// Mitsubishi GX Works2 project: LABB1.2   PLC: FX3U/FX3UC

// global labels: Global1
VAR_GLOBAL
  VK_VAN1 AT X000 : BOOL;  (* VÅNINGSKNAPP *)
  VK_VAN2 AT X001 : BOOL;
  VK_VAN3 AT X002 : BOOL;
  VK_VAN4 AT X003 : BOOL;
  GL_VAN1 AT X004 : BOOL;  (* POSITIONSREGISTER *)
  GL_VAN2 AT X005 : BOOL;
  GL_VAN3 AT X006 : BOOL;
  GL_VAN4 AT X007 : BOOL;
  HK_VAN1 AT X010 : BOOL;
  HK_VAN2 AT X011 : BOOL;  (* HISSKNAPP *)
  HK_VAN3 AT X012 : BOOL;
  HK_VAN4 AT X013 : BOOL;
  HL_VAN1 AT Y000 : BOOL;  (* HISSLAMPA *)
  HL_VAN2 AT Y001 : BOOL;
  HL_VAN3 AT Y002 : BOOL;
  HL_VAN4 AT Y003 : BOOL;
  VL_VAN1 AT Y004 : BOOL;  (* VÅNINGSLAMPA *)
  VL_VAN2 AT Y005 : BOOL;
  VL_VAN3 AT Y006 : BOOL;
  VL_VAN4 AT Y007 : BOOL;
  Motor_upp AT Y010 : BOOL;  (* HISS UPP *)
  Motor_ner AT Y011 : BOOL;  (* HISS NER *)
  PULS_1Hz AT M8013 : BOOL;  (* KLOCKFREKVENS FÖR VL *)
  ALARM_10Hz AT M8012 : BOOL;  (* ALARMFREKVENS *)
  TEMP AT Y012 : BOOL;  (* TEMP *)
  SWITCH AT Y013 : BOOL;  (* SWITCH *)
  SEC AT D100 : INT;
  MINUTE AT D101 : INT;
  TIMMAR AT D102 : INT;
  DAG AT D103 : INT;
  MANAD AT D104 : INT;
  AR AT D105 : INT;
  SEC2 AT D110 : INT;
  MINUTE2 AT D111 : INT;
  TIMMAR2 AT D112 : INT;
  DAG2 AT D113 : INT;
  MANAD2 AT D114 : INT;
  AR2 AT D115 : INT;
END_VAR

PROGRAM MAIN
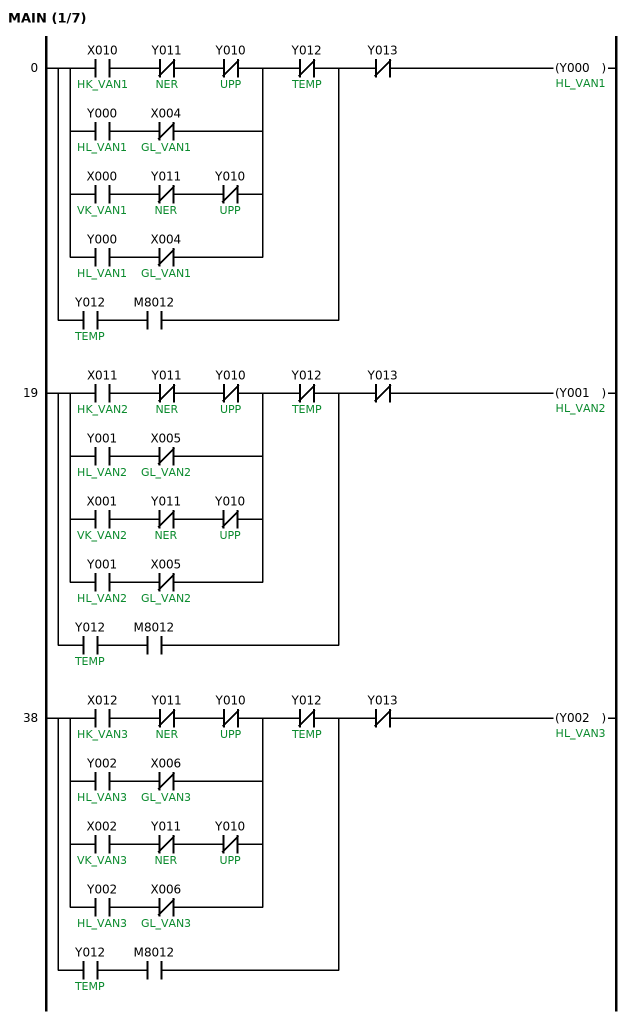
0     LD      X010  ; HK_VAN1
      ANI     Y011  ; NER
      ANI     Y010  ; UPP
      LD      Y000  ; HL_VAN1
      ANI     X004  ; GL_VAN1
      ORB
      LD      X000  ; VK_VAN1
      ANI     Y011  ; NER
      ANI     Y010  ; UPP
      ORB
      LD      Y000  ; HL_VAN1
      ANI     X004  ; GL_VAN1
      ORB
      ANI     Y012  ; TEMP
      LD      Y012  ; TEMP
      AND     M8012
      ORB
      ANI     Y013
      OUT     Y000  ; HL_VAN1
19    LD      X011  ; HK_VAN2
      ANI     Y011  ; NER
      ANI     Y010  ; UPP
      LD      Y001  ; HL_VAN2
      ANI     X005  ; GL_VAN2
      ORB
      LD      X001  ; VK_VAN2
      ANI     Y011  ; NER
      ANI     Y010  ; UPP
      ORB
      LD      Y001  ; HL_VAN2
      ANI     X005  ; GL_VAN2
      ORB
      ANI     Y012  ; TEMP
      LD      Y012  ; TEMP
      AND     M8012
      ORB
      ANI     Y013
      OUT     Y001  ; HL_VAN2
38    LD      X012  ; HK_VAN3
      ANI     Y011  ; NER
      ANI     Y010  ; UPP
      LD      Y002  ; HL_VAN3
      ANI     X006  ; GL_VAN3
      ORB
      LD      X002  ; VK_VAN3
      ANI     Y011  ; NER
      ANI     Y010  ; UPP
      ORB
      LD      Y002  ; HL_VAN3
      ANI     X006  ; GL_VAN3
      ORB
      ANI     Y012  ; TEMP
      LD      Y012  ; TEMP
      AND     M8012
      ORB
      ANI     Y013
      OUT     Y002  ; HL_VAN3
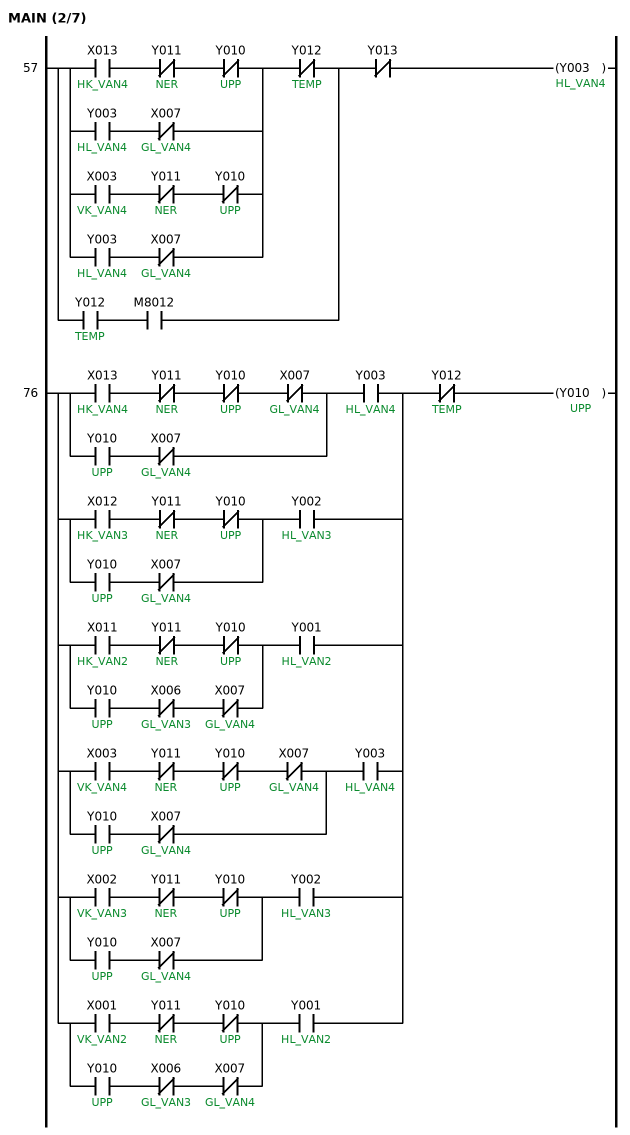
57    LD      X013  ; HK_VAN4
      ANI     Y011  ; NER
      ANI     Y010  ; UPP
      LD      Y003  ; HL_VAN4
      ANI     X007  ; GL_VAN4
      ORB
      LD      X003  ; VK_VAN4
      ANI     Y011  ; NER
      ANI     Y010  ; UPP
      ORB
      LD      Y003  ; HL_VAN4
      ANI     X007  ; GL_VAN4
      ORB
      ANI     Y012  ; TEMP
      LD      Y012  ; TEMP
      AND     M8012
      ORB
      ANI     Y013
      OUT     Y003  ; HL_VAN4
76    LD      X013  ; HK_VAN4
      ANI     Y011  ; NER
      ANI     Y010  ; UPP
      ANI     X007  ; GL_VAN4
      LD      Y010  ; UPP
      ANI     X007  ; GL_VAN4
      ORB
      AND     Y003  ; HL_VAN4
      LD      X012  ; HK_VAN3
      ANI     Y011  ; NER
      ANI     Y010  ; UPP
      LD      Y010  ; UPP
      ANI     X007  ; GL_VAN4
      ORB
      AND     Y002  ; HL_VAN3
      ORB
      LD      X011  ; HK_VAN2
      ANI     Y011  ; NER
      ANI     Y010  ; UPP
      LD      Y010  ; UPP
      ANI     X006  ; GL_VAN3
      ANI     X007  ; GL_VAN4
      ORB
      AND     Y001  ; HL_VAN2
      ORB
      LD      X003  ; VK_VAN4
      ANI     Y011  ; NER
      ANI     Y010  ; UPP
      ANI     X007  ; GL_VAN4
      LD      Y010  ; UPP
      ANI     X007  ; GL_VAN4
      ORB
      AND     Y003  ; HL_VAN4
      ORB
      LD      X002  ; VK_VAN3
      ANI     Y011  ; NER
      ANI     Y010  ; UPP
      LD      Y010  ; UPP
      ANI     X007  ; GL_VAN4
      ORB
      AND     Y002  ; HL_VAN3
      ORB
      LD      X001  ; VK_VAN2
      ANI     Y011  ; NER
      ANI     Y010  ; UPP
      LD      Y010  ; UPP
      ANI     X006  ; GL_VAN3
      ANI     X007  ; GL_VAN4
      ORB
      AND     Y001  ; HL_VAN2
      ORB
      ANI     Y012  ; TEMP
      OUT     Y010  ; UPP
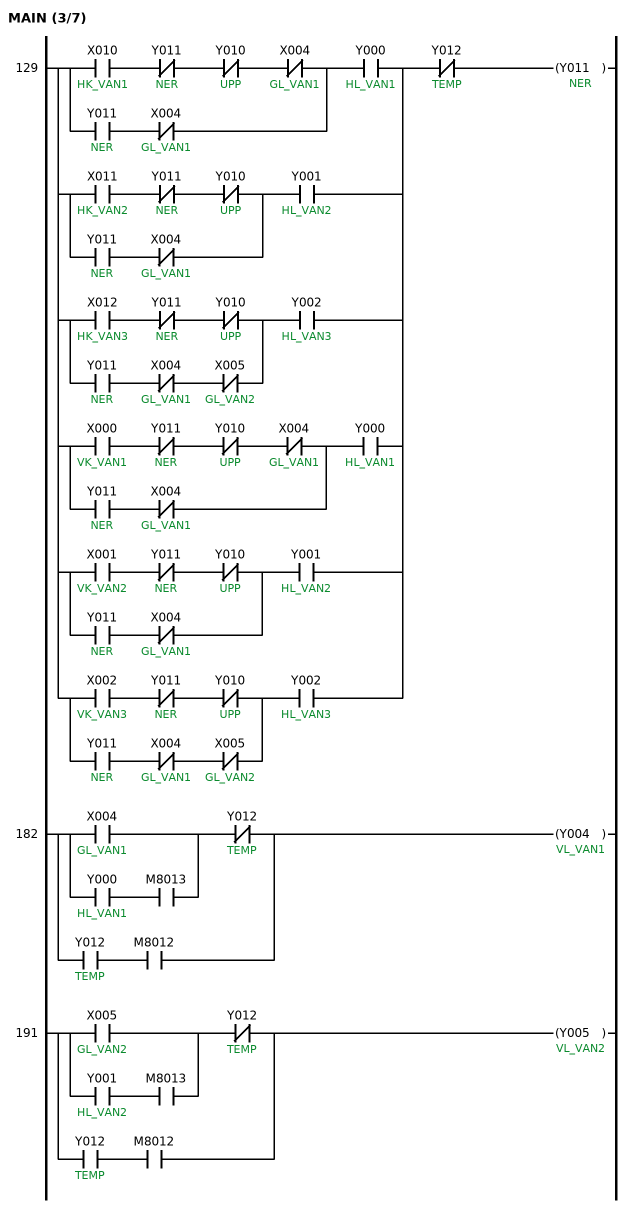
129   LD      X010  ; HK_VAN1
      ANI     Y011  ; NER
      ANI     Y010  ; UPP
      ANI     X004  ; GL_VAN1
      LD      Y011  ; NER
      ANI     X004  ; GL_VAN1
      ORB
      AND     Y000  ; HL_VAN1
      LD      X011  ; HK_VAN2
      ANI     Y011  ; NER
      ANI     Y010  ; UPP
      LD      Y011  ; NER
      ANI     X004  ; GL_VAN1
      ORB
      AND     Y001  ; HL_VAN2
      ORB
      LD      X012  ; HK_VAN3
      ANI     Y011  ; NER
      ANI     Y010  ; UPP
      LD      Y011  ; NER
      ANI     X004  ; GL_VAN1
      ANI     X005  ; GL_VAN2
      ORB
      AND     Y002  ; HL_VAN3
      ORB
      LD      X000  ; VK_VAN1
      ANI     Y011  ; NER
      ANI     Y010  ; UPP
      ANI     X004  ; GL_VAN1
      LD      Y011  ; NER
      ANI     X004  ; GL_VAN1
      ORB
      AND     Y000  ; HL_VAN1
      ORB
      LD      X001  ; VK_VAN2
      ANI     Y011  ; NER
      ANI     Y010  ; UPP
      LD      Y011  ; NER
      ANI     X004  ; GL_VAN1
      ORB
      AND     Y001  ; HL_VAN2
      ORB
      LD      X002  ; VK_VAN3
      ANI     Y011  ; NER
      ANI     Y010  ; UPP
      LD      Y011  ; NER
      ANI     X004  ; GL_VAN1
      ANI     X005  ; GL_VAN2
      ORB
      AND     Y002  ; HL_VAN3
      ORB
      ANI     Y012  ; TEMP
      OUT     Y011  ; NER
182   LD      X004  ; GL_VAN1
      LD      Y000  ; HL_VAN1
      AND     M8013
      ORB
      ANI     Y012  ; TEMP
      LD      Y012  ; TEMP
      AND     M8012
      ORB
      OUT     Y004  ; VL_VAN1
191   LD      X005  ; GL_VAN2
      LD      Y001  ; HL_VAN2
      AND     M8013
      ORB
      ANI     Y012  ; TEMP
      LD      Y012  ; TEMP
      AND     M8012
      ORB
      OUT     Y005  ; VL_VAN2
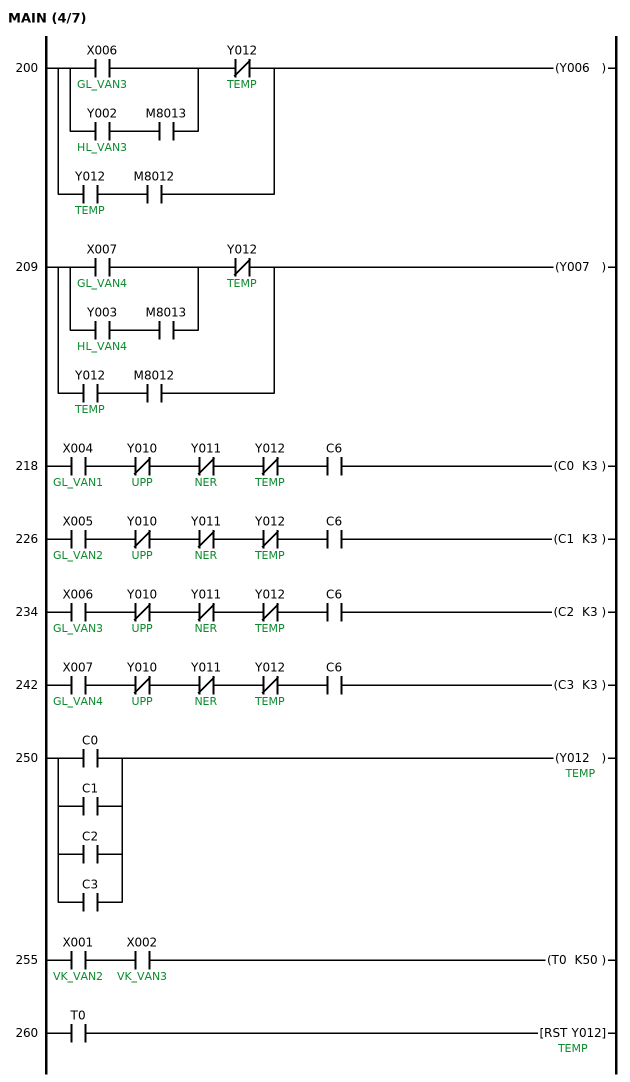
200   LD      X006  ; GL_VAN3
      LD      Y002  ; HL_VAN3
      AND     M8013
      ORB
      ANI     Y012  ; TEMP
      LD      Y012  ; TEMP
      AND     M8012
      ORB
      OUT     Y006
209   LD      X007  ; GL_VAN4
      LD      Y003  ; HL_VAN4
      AND     M8013
      ORB
      ANI     Y012  ; TEMP
      LD      Y012  ; TEMP
      AND     M8012
      ORB
      OUT     Y007
218   LD      X004  ; GL_VAN1
      ANI     Y010  ; UPP
      ANI     Y011  ; NER
      ANI     Y012  ; TEMP
      AND     C6
      OUT     C0 K3
226   LD      X005  ; GL_VAN2
      ANI     Y010  ; UPP
      ANI     Y011  ; NER
      ANI     Y012  ; TEMP
      AND     C6
      OUT     C1 K3
234   LD      X006  ; GL_VAN3
      ANI     Y010  ; UPP
      ANI     Y011  ; NER
      ANI     Y012  ; TEMP
      AND     C6
      OUT     C2 K3
242   LD      X007  ; GL_VAN4
      ANI     Y010  ; UPP
      ANI     Y011  ; NER
      ANI     Y012  ; TEMP
      AND     C6
      OUT     C3 K3
250   LD      C0
      OR      C1
      OR      C2
      OR      C3
      OUT     Y012  ; TEMP
255   LD      X001  ; VK_VAN2
      AND     X002  ; VK_VAN3
      OUT     T0 K50
260   LD      T0
      RST     Y012  ; TEMP
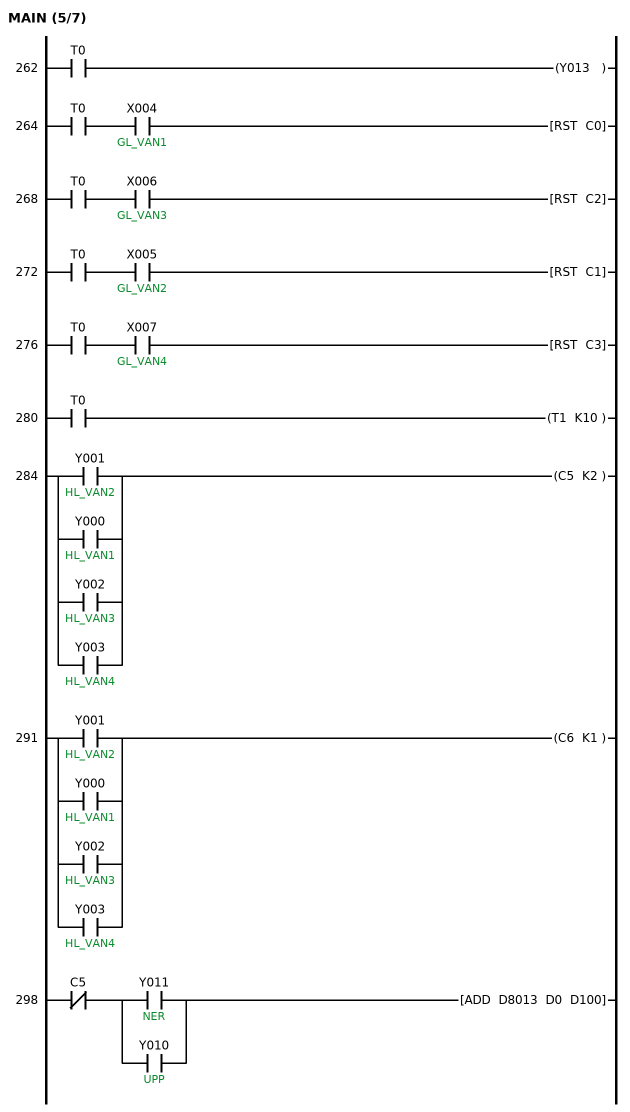
262   LD      T0
      OUT     Y013
264   LD      T0
      AND     X004  ; GL_VAN1
      RST     C0
268   LD      T0
      AND     X006  ; GL_VAN3
      RST     C2
272   LD      T0
      AND     X005  ; GL_VAN2
      RST     C1
276   LD      T0
      AND     X007  ; GL_VAN4
      RST     C3
280   LD      T0
      OUT     T1 K10
284   LD      Y001  ; HL_VAN2
      OR      Y000  ; HL_VAN1
      OR      Y002  ; HL_VAN3
      OR      Y003  ; HL_VAN4
      OUT     C5 K2
291   LD      Y001  ; HL_VAN2
      OR      Y000  ; HL_VAN1
      OR      Y002  ; HL_VAN3
      OR      Y003  ; HL_VAN4
      OUT     C6 K1
298   LDI     C5
      LD      Y011  ; NER
      OR      Y010  ; UPP
      ANB
      ADD     D8013 D0 D100
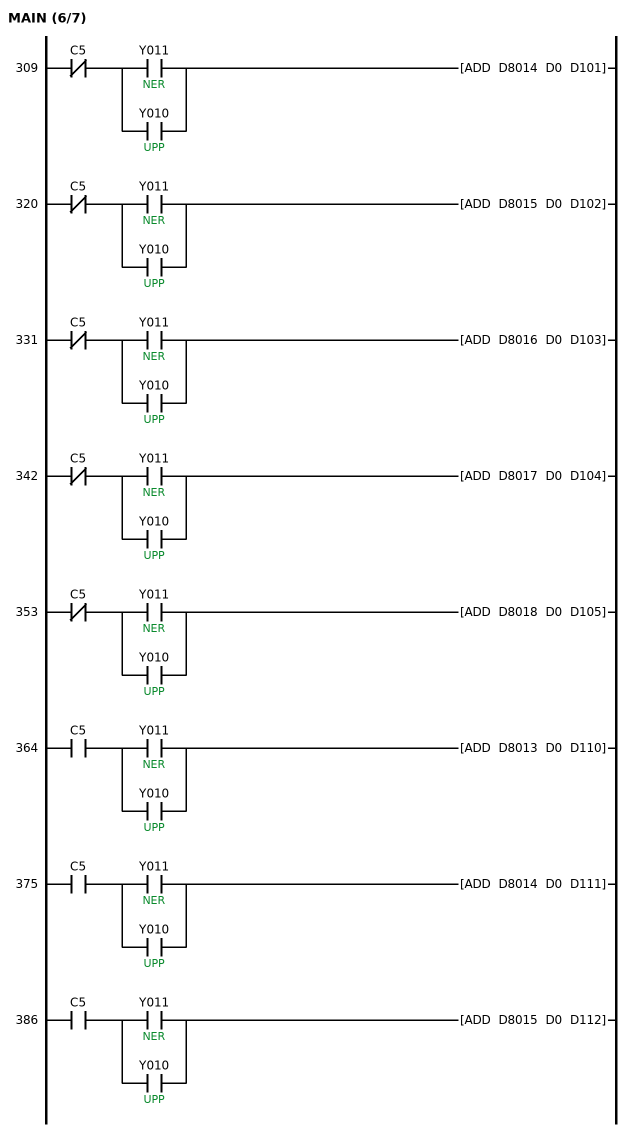
309   LDI     C5
      LD      Y011  ; NER
      OR      Y010  ; UPP
      ANB
      ADD     D8014 D0 D101
320   LDI     C5
      LD      Y011  ; NER
      OR      Y010  ; UPP
      ANB
      ADD     D8015 D0 D102
331   LDI     C5
      LD      Y011  ; NER
      OR      Y010  ; UPP
      ANB
      ADD     D8016 D0 D103
342   LDI     C5
      LD      Y011  ; NER
      OR      Y010  ; UPP
      ANB
      ADD     D8017 D0 D104
353   LDI     C5
      LD      Y011  ; NER
      OR      Y010  ; UPP
      ANB
      ADD     D8018 D0 D105
364   LD      C5
      LD      Y011  ; NER
      OR      Y010  ; UPP
      ANB
      ADD     D8013 D0 D110
375   LD      C5
      LD      Y011  ; NER
      OR      Y010  ; UPP
      ANB
      ADD     D8014 D0 D111
386   LD      C5
      LD      Y011  ; NER
      OR      Y010  ; UPP
      ANB
      ADD     D8015 D0 D112
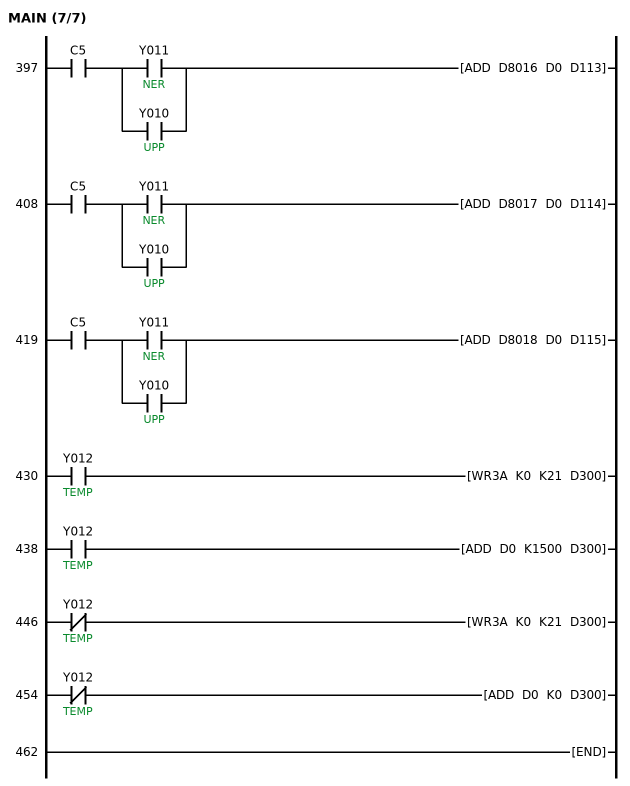
397   LD      C5
      LD      Y011  ; NER
      OR      Y010  ; UPP
      ANB
      ADD     D8016 D0 D113
408   LD      C5
      LD      Y011  ; NER
      OR      Y010  ; UPP
      ANB
      ADD     D8017 D0 D114
419   LD      C5
      LD      Y011  ; NER
      OR      Y010  ; UPP
      ANB
      ADD     D8018 D0 D115
430   LD      Y012  ; TEMP
      WR3A    K0 K21 D300
438   LD      Y012  ; TEMP
      ADD     D0 K1500 D300
446   LDI     Y012  ; TEMP
      WR3A    K0 K21 D300
454   LDI     Y012  ; TEMP
      ADD     D0 K0 D300
462   END
END_PROGRAM
